(* CODESYS project MC500.project
   Title: MC500
   CompiledLibraryCompatibilityVersion: LeadSysStudio V3.5 SP15 Patch 4

Project tree, tasks and I/O mapping:
  Device : MC508, Leadshine Technology Co., Ltd., order no. 508101, version 3.5.15.40
      settings: RetainMode = 0; RetainStartAddr = 20480; RetainEndAddr = 524288; RetainSize = 524288
    application Application
      libraries: Standard, * (System); VisuDialogs, * (System)
      task EtherCAT_Master_Leadshine_A (cyclic, interval 2000 µs, priority 0) calls EtherCAT_Master_Leadshine_A.EtherCAT_Task [EtherCAT_Master_Leadshine_A.EtherCAT_Task], main
      program main [ST]: initialize, motion, gear, io, tap, index, work, WRAP
      visualisation Visualization
      trace Trace (task EtherCAT_Master_Leadshine_A): main.gear_data.trace_master, main.gear_data.trace_slave, main.gear_data.trace_delta
      data type GearData
      data type IOTestData
      data type TapData
      data type IndexData
      data type WorkData
      Symbols
      data type ButtonData
    Device Diagnose
    Network Configuration
      LocalBus Config
    Resource Usage
    SoftMotion General Axis Pool
    High_Speed_IO_Module : High Speed IO, Leadshine Technology Co., Ltd., version 3.5.15.40
        unmapped channels: Genral_IO_IN, Genral_IO_Out
    LocalBus_Master_Module : LocalBus Master, Leadshine Technology Co., Ltd., version 3.5.15.40
    EtherCAT_Master_Leadshine_A : EtherCAT Master SoftMotion, 3S - Smart Software Solutions GmbH, version 3.5.15.30
        settings: MasterCycleTime = 2000; NetworkName = 'ecat'; SelectNetworkByName = False; SrcAddress1 = 10; SrcAddress2 = 889192738
      AxisX : XINJE-DS5C EtherCAT(CoE) Drive Rev2.0 v3.7.30, Xinje Electronics, Inc., order no. XINJE-DS5C CoE Drive Rev2.0, version Revision=16#02040608
          settings: Number of Inputs = 6; Number of Infos about Inputs = 6; EnableExpertSettings = True; StationAlias = 1; DeviceIdenticationADO = 0; DeviceIdenticationMode = 0; Sync.Length = 17; FMMU.Length = 17; DC sync0 cycletime = 2000; DC sync1 cycletime = 2000; Number of SDO = 5; Interpolation time period.Value = 2; Homing method.Index = 16#0000; Homing method.Subindex = 16#00; Homing method.Size = 0; Homing method.AbortIfError = FALSE; Homing method.JumpToLine = FALSE; Homing method.Line = 0; Homing method.CompleteAccess = False; Homing method.Index = 16#0000; Homing method.Subindex = 16#00; Homing method.Size = 0; Homing method.AbortIfError = FALSE; Homing method.JumpToLine = FALSE; Homing method.Line = 0; Homing method.CompleteAccess = False; RxTxPdo.NumberofEntries = 6; RxTxPdo.Index = 16#1A00; RxTxPdo.DependOnSlot = False; RxTxPdo.DependOnSlotGroup = False; RxTxPdo.OverwrittenByModule = False; Status Word.Offset = 0; Status Word.DependOnSlot = False; Status Word.DependOnSlotGroup = False; ActualPosition.Offset = 0; ActualPosition.DependOnSlot = False; ActualPosition.DependOnSlotGroup = False; Velocity actual value.Offset = 0; Velocity actual value.DependOnSlot = False; Velocity actual value.DependOnSlotGroup = False;
            ActualTorque.Offset = 0; ActualTorque.DependOnSlot = False; ActualTorque.DependOnSlotGroup = False; ModeOfOperationDisplay.Offset = 0; ModeOfOperationDisplay.DependOnSlot = False; ModeOfOperationDisplay.DependOnSlotGroup = False; Index = 16#5000; SubIndex = 0; Size = 32; Offset = 0; DependOnSlot = False; DependOnSlotGroup = False; Status Word.Default = ''; Status Word.Comment = ''; ActualPosition.Default = ''; ActualPosition.Comment = ''; Velocity actual value.Default = ''; Velocity actual value.Comment = ''; ActualTorque.Default = ''; ActualTorque.Comment = ''; ModeOfOperationDisplay.Default = ''; ModeOfOperationDisplay.Comment = ''; Name = 'Encode Single Position'; DataType = 'DINT'; Default = ''; Comment = ''
          unmapped channels: Control Word, TargetPosition, TargetVelocity, TargetTorque, ModeOfOperation, Status Word, ActualPosition, Velocity actual value, %IW8 ActualTorque, ModeOfOperationDisplay, %ID5 Encode Single Position
        AX : Axis, 3S - Smart Software Solutions GmbH, order no. 0, version 4.6.1.0
            settings: wDriveID = 0; dwRatioTechUnitsDenom = 16384; iRatioTechUnitsNum = 625; fSWLimitPositive = 5000.0; Number of pulses for one revolution = 1; The displacement for one revolution of the workbench = 1; Gear ratio molecule = 131072; Gear ratio denominator = 5000; ScalingIncs = 1; ScalingMotorTurns2 = 131072; ScalingGearOutput1 = 5000; AdrOffset_8010 = 4; BitOffset_8010 = 0; BitLength_8010 = 16; Address_8010 = '%QW2'; Type_8010 = 'UINT'; AddressPointer_8010 = ADR(%QW2); AdrOffset_8020 = 8; BitOffset_8020 = 0; BitLength_8020 = 32; Address_8020 = '%QD2'; Type_8020 = 'DINT'; AddressPointer_8020 = ADR(%QD2); AdrOffset_8030 = 12; BitOffset_8030 = 0; BitLength_8030 = 32; Address_8030 = '%QD3'; Type_8030 = 'DINT'; AddressPointer_8030 = ADR(%QD3); AdrOffset_8040 = 16; BitOffset_8040 = 0; BitLength_8040 = 16; Address_8040 = '%QW8'; Type_8040 = 'INT'; AddressPointer_8040 = ADR(%QW8); AdrOffset_8050 = 18; BitOffset_8050 = 0; BitLength_8050 = 8; Address_8050 = '%QB18'; Type_8050 = 'SINT';
              AddressPointer_8050 = ADR(%QB18); AdrOffset_8060 = 4294967295; BitOffset_8060 = 0; BitLength_8060 = 0; Address_8060 = ''; Type_8060 = ''; AddressPointer_8060 = 0; AdrOffset_8070 = 4294967295; BitOffset_8070 = 0; BitLength_8070 = 0; Address_8070 = ''; Type_8070 = ''; AddressPointer_8070 = 0; AdrOffset_8080 = 4294967295; BitOffset_8080 = 0; BitLength_8080 = 0; Address_8080 = ''; Type_8080 = ''; AddressPointer_8080 = 0; AdrOffset_8090 = 4294967295; BitOffset_8090 = 0; BitLength_8090 = 0; Address_8090 = ''; Type_8090 = ''; AddressPointer_8090 = 0; AdrOffset_8510 = 4; BitOffset_8510 = 0; BitLength_8510 = 16; Address_8510 = '%IW2'; Type_8510 = 'UINT'; AddressPointer_8510 = ADR(%IW2); AdrOffset_8520 = 8; BitOffset_8520 = 0; BitLength_8520 = 32; Address_8520 = '%ID2'; Type_8520 = 'DINT'; AddressPointer_8520 = ADR(%ID2); AdrOffset_8530 = 12; BitOffset_8530 = 0; BitLength_8530 = 32;
              Address_8530 = '%ID3'; Type_8530 = 'DINT'; AddressPointer_8530 = ADR(%ID3); AdrOffset_8540 = 16; BitOffset_8540 = 0; BitLength_8540 = 16; Address_8540 = '%IW8'; Type_8540 = 'INT'; AddressPointer_8540 = ADR(%IW8); AdrOffset_8550 = 18; BitOffset_8550 = 0; BitLength_8550 = 8; Address_8550 = '%IB18'; Type_8550 = 'SINT'; AddressPointer_8550 = ADR(%IB18); AdrOffset_8560 = 4294967295; BitOffset_8560 = 0; BitLength_8560 = 0; Address_8560 = ''; Type_8560 = ''; AddressPointer_8560 = 0; AdrOffset_8570 = 4294967295; BitOffset_8570 = 0; BitLength_8570 = 0; Address_8570 = ''; Type_8570 = ''; AddressPointer_8570 = 0; AdrOffset_8580 = 4294967295; BitOffset_8580 = 0; BitLength_8580 = 0; Address_8580 = ''; Type_8580 = ''; AddressPointer_8580 = 0; AdrOffset_8590 = 4294967295; BitOffset_8590 = 0; BitLength_8590 = 0; Address_8590 = ''; Type_8590 = ''; AddressPointer_8590 = 0; AdrOffset_8600 = 4294967295;
              BitOffset_8600 = 0; BitLength_8600 = 0; Address_8600 = ''; Type_8600 = ''; AddressPointer_8600 = 0; AdrOffset_8600 = 4294967295; BitOffset_8600 = 0; BitLength_8600 = 0; Address_8610 = ''; Type_8610 = ''; AddressPointer_8610 = 0; AdrOffset_8620 = 4294967295; BitOffset_8620 = 0; BitLength_8620 = 0; Address_8620 = ''; Type_8620 = ''; AddressPointer_8620 = 0
      AxisY : XINJE-DS5C EtherCAT(CoE) Drive Rev2.0 v3.7.30, Xinje Electronics, Inc., order no. XINJE-DS5C CoE Drive Rev2.0, version Revision=16#02040608
          settings: Number of Inputs = 6; Number of Infos about Inputs = 6; EnableExpertSettings = True; StationAlias = 2; DeviceIdenticationADO = 0; DeviceIdenticationMode = 0; Sync.Length = 17; FMMU.Length = 17; DC sync0 cycletime = 2000; DC sync1 cycletime = 2000; Number of SDO = 5; Interpolation time period.Value = 2; Homing method.Index = 16#0000; Homing method.Subindex = 16#00; Homing method.Size = 0; Homing method.AbortIfError = FALSE; Homing method.JumpToLine = FALSE; Homing method.Line = 0; Homing method.CompleteAccess = False; Homing method.Index = 16#0000; Homing method.Subindex = 16#00; Homing method.Size = 0; Homing method.AbortIfError = FALSE; Homing method.JumpToLine = FALSE; Homing method.Line = 0; Homing method.CompleteAccess = False; RxTxPdo.NumberofEntries = 6; RxTxPdo.Index = 16#1A00; RxTxPdo.DependOnSlot = False; RxTxPdo.DependOnSlotGroup = False; RxTxPdo.OverwrittenByModule = False; Status Word.Offset = 0; Status Word.DependOnSlot = False; Status Word.DependOnSlotGroup = False; ActualPosition.Offset = 0; ActualPosition.DependOnSlot = False; ActualPosition.DependOnSlotGroup = False; Velocity actual value.Offset = 0; Velocity actual value.DependOnSlot = False; Velocity actual value.DependOnSlotGroup = False;
            ActualTorque.Offset = 0; ActualTorque.DependOnSlot = False; ActualTorque.DependOnSlotGroup = False; ModeOfOperationDisplay.Offset = 0; ModeOfOperationDisplay.DependOnSlot = False; ModeOfOperationDisplay.DependOnSlotGroup = False; Index = 16#5000; SubIndex = 0; Size = 32; Offset = 0; DependOnSlot = False; DependOnSlotGroup = False; Status Word.Default = ''; Status Word.Comment = ''; ActualPosition.Default = ''; ActualPosition.Comment = ''; Velocity actual value.Default = ''; Velocity actual value.Comment = ''; ActualTorque.Default = ''; ActualTorque.Comment = ''; ModeOfOperationDisplay.Default = ''; ModeOfOperationDisplay.Comment = ''; Name = 'Encode Single Position'; DataType = 'DINT'; Default = ''; Comment = ''
          unmapped channels: Control Word, TargetPosition, TargetVelocity, TargetTorque, ModeOfOperation, Status Word, ActualPosition, Velocity actual value, %IW18 ActualTorque, ModeOfOperationDisplay, %ID10 Encode Single Position
        AY : Axis, 3S - Smart Software Solutions GmbH, order no. 0, version 4.6.1.0
            settings: dwRatioTechUnitsDenom = 16384; iRatioTechUnitsNum = 125; Number of pulses for one revolution = 1; The displacement for one revolution of the workbench = 1; Gear ratio molecule = 131072; Gear ratio denominator = 1000; ScalingIncs = 1; ScalingMotorTurns2 = 131072; ScalingGearOutput1 = 1000; AdrOffset_8010 = 20; BitOffset_8010 = 0; BitLength_8010 = 16; Address_8010 = '%QW10'; Type_8010 = 'UINT'; AddressPointer_8010 = ADR(%QW10); AdrOffset_8020 = 24; BitOffset_8020 = 0; BitLength_8020 = 32; Address_8020 = '%QD6'; Type_8020 = 'DINT'; AddressPointer_8020 = ADR(%QD6); AdrOffset_8030 = 28; BitOffset_8030 = 0; BitLength_8030 = 32; Address_8030 = '%QD7'; Type_8030 = 'DINT'; AddressPointer_8030 = ADR(%QD7); AdrOffset_8040 = 32; BitOffset_8040 = 0; BitLength_8040 = 16; Address_8040 = '%QW16'; Type_8040 = 'INT'; AddressPointer_8040 = ADR(%QW16); AdrOffset_8050 = 34; BitOffset_8050 = 0; BitLength_8050 = 8; Address_8050 = '%QB34'; Type_8050 = 'SINT'; AddressPointer_8050 = ADR(%QB34); AdrOffset_8060 = 4294967295;
              BitOffset_8060 = 0; BitLength_8060 = 0; Address_8060 = ''; Type_8060 = ''; AddressPointer_8060 = 0; AdrOffset_8070 = 4294967295; BitOffset_8070 = 0; BitLength_8070 = 0; Address_8070 = ''; Type_8070 = ''; AddressPointer_8070 = 0; AdrOffset_8080 = 4294967295; BitOffset_8080 = 0; BitLength_8080 = 0; Address_8080 = ''; Type_8080 = ''; AddressPointer_8080 = 0; AdrOffset_8090 = 4294967295; BitOffset_8090 = 0; BitLength_8090 = 0; Address_8090 = ''; Type_8090 = ''; AddressPointer_8090 = 0; AdrOffset_8510 = 24; BitOffset_8510 = 0; BitLength_8510 = 16; Address_8510 = '%IW12'; Type_8510 = 'UINT'; AddressPointer_8510 = ADR(%IW12); AdrOffset_8520 = 28; BitOffset_8520 = 0; BitLength_8520 = 32; Address_8520 = '%ID7'; Type_8520 = 'DINT'; AddressPointer_8520 = ADR(%ID7); AdrOffset_8530 = 32; BitOffset_8530 = 0; BitLength_8530 = 32; Address_8530 = '%ID8'; Type_8530 = 'DINT';
              AddressPointer_8530 = ADR(%ID8); AdrOffset_8540 = 36; BitOffset_8540 = 0; BitLength_8540 = 16; Address_8540 = '%IW18'; Type_8540 = 'INT'; AddressPointer_8540 = ADR(%IW18); AdrOffset_8550 = 38; BitOffset_8550 = 0; BitLength_8550 = 8; Address_8550 = '%IB38'; Type_8550 = 'SINT'; AddressPointer_8550 = ADR(%IB38); AdrOffset_8560 = 4294967295; BitOffset_8560 = 0; BitLength_8560 = 0; Address_8560 = ''; Type_8560 = ''; AddressPointer_8560 = 0; AdrOffset_8570 = 4294967295; BitOffset_8570 = 0; BitLength_8570 = 0; Address_8570 = ''; Type_8570 = ''; AddressPointer_8570 = 0; AdrOffset_8580 = 4294967295; BitOffset_8580 = 0; BitLength_8580 = 0; Address_8580 = ''; Type_8580 = ''; AddressPointer_8580 = 0; AdrOffset_8590 = 4294967295; BitOffset_8590 = 0; BitLength_8590 = 0; Address_8590 = ''; Type_8590 = ''; AddressPointer_8590 = 0; AdrOffset_8600 = 4294967295; BitOffset_8600 = 0; BitLength_8600 = 0;
              Address_8600 = ''; Type_8600 = ''; AddressPointer_8600 = 0; AdrOffset_8600 = 4294967295; BitOffset_8600 = 0; BitLength_8600 = 0; Address_8610 = ''; Type_8610 = ''; AddressPointer_8610 = 0; AdrOffset_8620 = 4294967295; BitOffset_8620 = 0; BitLength_8620 = 0; Address_8620 = ''; Type_8620 = ''; AddressPointer_8620 = 0
      AxisZ : XINJE-DS5C1 EtherCAT(CoE) Drive Rev4.0 v3.7.70, Xinje Electronics, Inc., order no. XINJE-DS5C1 CoE Drive Rev4.0, version Revision=16#20201207
          settings: Number of Inputs = 6; Number of Infos about Inputs = 6; EnableExpertSettings = True; StationAlias = 3; DeviceIdenticationADO = 0; DeviceIdenticationMode = 0; Sync.Length = 17; FMMU.Length = 17; DC sync0 cycletime = 2000; DC sync1 cycletime = 2000; Number of SDO = 6; Interpolation time period.Value = 2; Homing method.Index = 16#0000; Homing method.Subindex = 16#00; Homing method.Size = 0; Homing method.AbortIfError = FALSE; Homing method.JumpToLine = FALSE; Homing method.Line = 0; Homing method.CompleteAccess = False; Homing method.Index = 16#0000; Homing method.Subindex = 16#00; Homing method.Size = 0; Homing method.AbortIfError = FALSE; Homing method.JumpToLine = FALSE; Homing method.Line = 0; Homing method.CompleteAccess = False; Homing method.Index = 16#0000; Homing method.Subindex = 16#00; Homing method.Size = 0; Homing method.AbortIfError = FALSE; Homing method.JumpToLine = FALSE; Homing method.Line = 0; Homing method.CompleteAccess = False; RxTxPdo.NumberofEntries = 6; RxTxPdo.Index = 16#1A00; RxTxPdo.DependOnSlot = False; RxTxPdo.DependOnSlotGroup = False; RxTxPdo.OverwrittenByModule = False; Status Word.Offset = 0; Status Word.DependOnSlot = False;
            Status Word.DependOnSlotGroup = False; ActualPosition.Offset = 0; ActualPosition.DependOnSlot = False; ActualPosition.DependOnSlotGroup = False; Velocity actual value.Offset = 0; Velocity actual value.DependOnSlot = False; Velocity actual value.DependOnSlotGroup = False; ActualTorque.Offset = 0; ActualTorque.DependOnSlot = False; ActualTorque.DependOnSlotGroup = False; ModeOfOperationDisplay.Offset = 0; ModeOfOperationDisplay.DependOnSlot = False; ModeOfOperationDisplay.DependOnSlotGroup = False; Index = 16#5000; SubIndex = 0; Size = 32; Offset = 0; DependOnSlot = False; DependOnSlotGroup = False; Status Word.Default = ''; Status Word.Comment = ''; ActualPosition.Default = ''; ActualPosition.Comment = ''; Velocity actual value.Default = ''; Velocity actual value.Comment = ''; ActualTorque.Default = ''; ActualTorque.Comment = ''; ModeOfOperationDisplay.Default = ''; ModeOfOperationDisplay.Comment = ''; Name = 'Encode Single Position'; DataType = 'DINT'; Default = ''; Comment = ''
          unmapped channels: Control Word, TargetPosition, TargetVelocity, TargetTorque, ModeOfOperation, Status Word, ActualPosition, Velocity actual value, %IW28 ActualTorque, ModeOfOperationDisplay, %ID15 Encode Single Position
        AZ : Axis, 3S - Smart Software Solutions GmbH, order no. 0, version 4.6.1.0
            settings: wDriveID = 2; dwRatioTechUnitsDenom = 1; iMovementType = 0; fPositionPeriod = 131072; Number of pulses for one revolution = 1; The displacement for one revolution of the workbench = 1; Gear ratio molecule = 1; Gear ratio denominator = 1; ScalingIncs = 1; AdrOffset_8010 = 36; BitOffset_8010 = 0; BitLength_8010 = 16; Address_8010 = '%QW18'; Type_8010 = 'UINT'; AddressPointer_8010 = ADR(%QW18); AdrOffset_8020 = 40; BitOffset_8020 = 0; BitLength_8020 = 32; Address_8020 = '%QD10'; Type_8020 = 'DINT'; AddressPointer_8020 = ADR(%QD10); AdrOffset_8030 = 44; BitOffset_8030 = 0; BitLength_8030 = 32; Address_8030 = '%QD11'; Type_8030 = 'DINT'; AddressPointer_8030 = ADR(%QD11); AdrOffset_8040 = 48; BitOffset_8040 = 0; BitLength_8040 = 16; Address_8040 = '%QW24'; Type_8040 = 'INT'; AddressPointer_8040 = ADR(%QW24); AdrOffset_8050 = 50; BitOffset_8050 = 0; BitLength_8050 = 8; Address_8050 = '%QB50'; Type_8050 = 'SINT'; AddressPointer_8050 = ADR(%QB50); AdrOffset_8060 = 4294967295;
              BitOffset_8060 = 0; BitLength_8060 = 0; Address_8060 = ''; Type_8060 = ''; AddressPointer_8060 = 0; AdrOffset_8070 = 4294967295; BitOffset_8070 = 0; BitLength_8070 = 0; Address_8070 = ''; Type_8070 = ''; AddressPointer_8070 = 0; AdrOffset_8080 = 4294967295; BitOffset_8080 = 0; BitLength_8080 = 0; Address_8080 = ''; Type_8080 = ''; AddressPointer_8080 = 0; AdrOffset_8090 = 4294967295; BitOffset_8090 = 0; BitLength_8090 = 0; Address_8090 = ''; Type_8090 = ''; AddressPointer_8090 = 0; AdrOffset_8510 = 44; BitOffset_8510 = 0; BitLength_8510 = 16; Address_8510 = '%IW22'; Type_8510 = 'UINT'; AddressPointer_8510 = ADR(%IW22); AdrOffset_8520 = 48; BitOffset_8520 = 0; BitLength_8520 = 32; Address_8520 = '%ID12'; Type_8520 = 'DINT'; AddressPointer_8520 = ADR(%ID12); AdrOffset_8530 = 52; BitOffset_8530 = 0; BitLength_8530 = 32; Address_8530 = '%ID13'; Type_8530 = 'DINT';
              AddressPointer_8530 = ADR(%ID13); AdrOffset_8540 = 56; BitOffset_8540 = 0; BitLength_8540 = 16; Address_8540 = '%IW28'; Type_8540 = 'INT'; AddressPointer_8540 = ADR(%IW28); AdrOffset_8550 = 58; BitOffset_8550 = 0; BitLength_8550 = 8; Address_8550 = '%IB58'; Type_8550 = 'SINT'; AddressPointer_8550 = ADR(%IB58); AdrOffset_8560 = 4294967295; BitOffset_8560 = 0; BitLength_8560 = 0; Address_8560 = ''; Type_8560 = ''; AddressPointer_8560 = 0; AdrOffset_8570 = 4294967295; BitOffset_8570 = 0; BitLength_8570 = 0; Address_8570 = ''; Type_8570 = ''; AddressPointer_8570 = 0; AdrOffset_8580 = 4294967295; BitOffset_8580 = 0; BitLength_8580 = 0; Address_8580 = ''; Type_8580 = ''; AddressPointer_8580 = 0; AdrOffset_8590 = 4294967295; BitOffset_8590 = 0; BitLength_8590 = 0; Address_8590 = ''; Type_8590 = ''; AddressPointer_8590 = 0; AdrOffset_8600 = 4294967295; BitOffset_8600 = 0; BitLength_8600 = 0;
              Address_8600 = ''; Type_8600 = ''; AddressPointer_8600 = 0; AdrOffset_8600 = 4294967295; BitOffset_8600 = 0; BitLength_8600 = 0; Address_8610 = ''; Type_8610 = ''; AddressPointer_8610 = 0; AdrOffset_8620 = 4294967295; BitOffset_8620 = 0; BitLength_8620 = 0; Address_8620 = ''; Type_8620 = ''; AddressPointer_8620 = 0
  text list GlobalTextList
*)

// Device/Application/GearData
TYPE GearData :
STRUCT
	state: INT;
	ratio_target: LREAL;
	ratio: LREAL;
	ratio_array: ARRAY[0..14] OF LREAL;
	ratio_array_index: INT;
	reset_gear_timer: TON;
	trace_master: LREAL;
	trace_slave: LREAL;
	trace_delta: LREAL;
END_STRUCT
END_TYPE

// Device/Application/IOTestData
TYPE IOTestData :
STRUCT
	out: WORD;
	out_timer: TON;
END_STRUCT
END_TYPE

// Device/Application/TapData
TYPE TapData :
STRUCT
	state: INT;
	home_torque: INT;
	home_feed_back: LREAL;
	home_feed_forward: LREAL;
	home_offset: LREAL;
	start_position: LREAL;
	end_position: LREAL;
	feed_rpm: LREAL;
	end_delay: INT;
	end_timer: TON;
	gear_type: INT;
END_STRUCT
END_TYPE

// Device/Application/IndexData
TYPE IndexData :
STRUCT
	state: INT;
	slot_count: INT;
	slot_index: INT;
	slot_index_nearest: INT;
	real_position: LREAL;
	soft_position: LREAL;
	target_position: LREAL;
	offset: LREAL;
	ecd_sing: LREAL;
	ecd_reso: LREAL;
	end_delay: INT;
	end_timer: TON;
	feed_rpm: LREAL;
	is_home_ing: BOOL;
	vibrate_distance: LREAL;
END_STRUCT
END_TYPE

// Device/Application/WorkData
TYPE WorkData :
STRUCT
	state: INT;
	stop_state: INT;
	end_delay: INT;
	end_timer: TON;
END_STRUCT
END_TYPE

// Device/Application/ButtonData
TYPE ButtonData :
STRUCT
	on: BOOL;
	off: BOOL;
END_STRUCT
END_TYPE

// Device/Application/main
PROGRAM main
VAR
	state: INT;
	AX_power: MC_Power;
	AY_power: MC_Power;
	AZ_power: MC_Power;
	AX_status: MC_ReadStatus;
	AY_status: MC_ReadStatus;
	AZ_status: MC_ReadStatus;
	AZ_stop: MC_Stop;
	AX_reset: MC_Reset;
	AY_reset: MC_Reset;
	AZ_reset: MC_Reset;
	AX_set_position: MC_SetPosition;
	AY_set_position: MC_SetPosition;
	AZ_set_position: MC_SetPosition;
	AZ_mabs: MC_MoveAbsolute;
	AX_read: SMC3_ETC_ReadParameter_CoE;
	AY_read: SMC3_ETC_ReadParameter_CoE;
	AZ_read: SMC3_ETC_ReadParameter_CoE;
	AX_write: SMC3_ETC_WriteParameter_CoE;
	AY_write: SMC3_ETC_WriteParameter_CoE;
	AZ_write: SMC3_ETC_WriteParameter_CoE;
	AX_follow: SMC_FollowPosition;
	AY_follow: SMC_FollowPosition;
	gear_data: GearData;
	AX_torque AT %IW8: INT;
	AY_torque AT %IW18: INT;
	AZ_torque AT %IW28: INT;
	AX_encoder_single AT %ID5: DINT;
	AY_encoder_single AT %ID10: DINT;
	AZ_encoder_single AT %ID15: DINT;
	AX_encoder_resolution: DINT;
	AY_encoder_resolution: DINT;
	AZ_encoder_resolution: DINT;
	io_test_data: IOTestData;
	index_data: IndexData;
	tap_data: TapData;
	work_data: WorkData;
	button_data: ButtonData;
END_VAR

CASE state OF
    0:
		initialize();
		state := state + 1;
	1:
		IF AX.wCommunicationState = 100 AND AY.wCommunicationState = 100 AND AZ.wCommunicationState = 100 THEN
			AX_power.Enable := TRUE;
			AY_power.Enable := TRUE;
			AZ_power.Enable := TRUE;
			AX_status.Enable := TRUE;
			AY_status.Enable := TRUE;
			AZ_status.Enable := TRUE;
			AX_power.bDriveStart := TRUE;
			AY_power.bDriveStart := TRUE;
			AZ_power.bDriveStart := TRUE;
			AX_power.bRegulatorOn := FALSE;
			AY_power.bRegulatorOn := FALSE;
			AZ_power.bRegulatorOn := FALSE;
			state := state + 1;
		END_IF
	2:
		gear_data.ratio_array_index := 0;
		work_data.state := 1;
		state := state + 1;
	3:
		io();
END_CASE

IF state >= 2 THEN
	gear();
	motion();
	index();
	tap();
	work();
END_IF

ACTION initialize:
gear_data.ratio_array_index := 0;
gear_data.ratio_array[0] := 0.5;
gear_data.ratio_array[1] := 1.0;
gear_data.ratio_array[2] := 1.5;
gear_data.ratio_array[3] := 2.0;
gear_data.ratio_array[4] := 2.5;
gear_data.ratio_array[5] := 3.0;
gear_data.ratio_array[6] := 3.5;
gear_data.ratio_array[7] := 4.0;
gear_data.ratio_array[8] := 4.5;
gear_data.ratio_array[9] := 5.0;
gear_data.ratio_array[10] := 10.0;
gear_data.ratio_array[11] := 15.0;
gear_data.ratio_array[12] := 20.0;
gear_data.ratio_array[13] := 25.0;
gear_data.ratio_array[14] := 50.0;
state := 0;
index_data.state := 0;
index_data.end_delay := 100;
index_data.slot_count := 8;
index_data.feed_rpm := 60.0;
index_data.vibrate_distance := 1.0 / 64.0;
tap_data.state := 0;
tap_data.end_delay := 25;
tap_data.home_torque := 200;
tap_data.home_feed_back := 2000.0;
tap_data.home_feed_forward := 3000.0;
tap_data.home_offset := 10_000.0;
tap_data.start_position := tap_data.home_offset;
tap_data.end_position := tap_data.home_offset + 7_000.0;
tap_data.feed_rpm := 800.0;
tap_data.gear_type := 1;
work_data.state := 0;
work_data.stop_state := 0;
work_data.end_delay := 25;
button_data.on := FALSE;
button_data.off := FALSE;
END_ACTION

ACTION motion:
IF AX.bCommunication AND AY.bCommunication AND AZ.bCommunication THEN
	//power
	AX_power( Axis:= AX, Enable:= , bRegulatorOn:= , bDriveStart:= , Status=> , bRegulatorRealState=> , bDriveStartRealState=> , Busy=> , Error=> , ErrorID=> );
	AY_power( Axis:= AY, Enable:= , bRegulatorOn:= , bDriveStart:= , Status=> , bRegulatorRealState=> , bDriveStartRealState=> , Busy=> , Error=> , ErrorID=> );
	AZ_power( Axis:= AZ, Enable:= , bRegulatorOn:= , bDriveStart:= , Status=> , bRegulatorRealState=> , bDriveStartRealState=> , Busy=> , Error=> , ErrorID=> );
	//status
	AX_status( Axis:= AX, Enable:= , Valid=> , Busy=> , Error=> , ErrorID=> , Disabled=> , Errorstop=> , Stopping=> , StandStill=> , DiscreteMotion=> , ContinuousMotion=> , SynchronizedMotion=> , Homing=> , ConstantVelocity=> , Accelerating=> , Decelerating=> , FBErrorOccured=> );
	AY_status( Axis:= AY, Enable:= , Valid=> , Busy=> , Error=> , ErrorID=> , Disabled=> , Errorstop=> , Stopping=> , StandStill=> , DiscreteMotion=> , ContinuousMotion=> , SynchronizedMotion=> , Homing=> , ConstantVelocity=> , Accelerating=> , Decelerating=> , FBErrorOccured=> );
	AZ_status( Axis:= AZ, Enable:= , Valid=> , Busy=> , Error=> , ErrorID=> , Disabled=> , Errorstop=> , Stopping=> , StandStill=> , DiscreteMotion=> , ContinuousMotion=> , SynchronizedMotion=> , Homing=> , ConstantVelocity=> , Accelerating=> , Decelerating=> , FBErrorOccured=> );
	//stop
	AZ_stop( Axis:= AZ, Execute:= , Deceleration:= , Jerk:= , Done=> , Busy=> , Error=> , ErrorID=> );
	//reset
	AX_reset( Axis:= AX, Execute:= , Done=> , Busy=> , Error=> , ErrorID=> );
	AY_reset( Axis:= AY, Execute:= , Done=> , Busy=> , Error=> , ErrorID=> );
	AZ_reset( Axis:= AZ, Execute:= , Done=> , Busy=> , Error=> , ErrorID=> );
	//set position
	AX_set_position( Axis:= AX, Execute:= , Position:= , Mode:= , Done=> , Busy=> , Error=> , ErrorID=> );
	AY_set_position( Axis:= AY, Execute:= , Position:= , Mode:= , Done=> , Busy=> , Error=> , ErrorID=> );
	AZ_set_position( Axis:= AZ, Execute:= , Position:= , Mode:= , Done=> , Busy=> , Error=> , ErrorID=> );
	//move absolute
	AZ_mabs( Axis:= AZ, Execute:= , Position:= , Velocity:= , Acceleration:= , Deceleration:= , Jerk:= , Direction:= , BufferMode:= , Done=> , Busy=> , Active=> , CommandAborted=> , Error=> , ErrorID=> );
	//read write
	AX_read( xExecute:= , xAbort:= , uiIndex:= , usiSubIndex:= , Axis:= AX, xDone=> , xBusy=> , xError=> , usiDataLength=> , dwValue=> , dwErrorCode=> , eError=> );
	AY_read( xExecute:= , xAbort:= , uiIndex:= , usiSubIndex:= , Axis:= AY, xDone=> , xBusy=> , xError=> , usiDataLength=> , dwValue=> , dwErrorCode=> , eError=> );
	AZ_read( xExecute:= , xAbort:= , uiIndex:= , usiSubIndex:= , Axis:= AZ, xDone=> , xBusy=> , xError=> , usiDataLength=> , dwValue=> , dwErrorCode=> , eError=> );
	AX_write( xExecute:= , xAbort:= , uiIndex:= , usiSubIndex:= , usiDataLength:= , dwValue:= , Axis:= AX, xDone=> , xBusy=> , xError=> , dwErrorCode=> , eError=> );
	AY_write( xExecute:= , xAbort:= , uiIndex:= , usiSubIndex:= , usiDataLength:= , dwValue:= , Axis:= AY, xDone=> , xBusy=> , xError=> , dwErrorCode=> , eError=> );
	AZ_write( xExecute:= , xAbort:= , uiIndex:= , usiSubIndex:= , usiDataLength:= , dwValue:= , Axis:= AZ, xDone=> , xBusy=> , xError=> , dwErrorCode=> , eError=> );
	//follow
	AX_follow( Axis:= AX, bExecute:= , fSetPosition:= , bBusy=> , bCommandAborted=> , bError=> , iErrorID=> );
	AY_follow( Axis:= AY, bExecute:= , fSetPosition:= , bBusy=> , bCommandAborted=> , bError=> , iErrorID=> );
END_IF
END_ACTION

ACTION gear:
gear_data.ratio_target := gear_data.ratio_array[gear_data.ratio_array_index];
gear_data.trace_master := AY.fActPosition;
gear_data.trace_slave := AX.fActPosition / gear_data.ratio;
gear_data.trace_delta := gear_data.trace_master - gear_data.trace_slave;
CASE gear_data.state OF
	0:
		gear_data.reset_gear_timer.IN := FALSE;
	1:
		AX_follow.bExecute := FALSE;
		AY_follow.bExecute := FALSE;
		AX_power.bRegulatorOn := FALSE;
		AY_power.bRegulatorOn := FALSE;
		gear_data.state := gear_data.state + 1;
	2:
		gear_data.reset_gear_timer(IN:= , PT:= , Q=> , ET=> );
		IF NOT gear_data.reset_gear_timer.IN THEN
			gear_data.reset_gear_timer.IN := TRUE;
			gear_data.reset_gear_timer.PT := INT_TO_TIME(100);
		END_IF
		IF gear_data.reset_gear_timer.Q THEN
			gear_data.reset_gear_timer.IN := FALSE;
			gear_data.state := gear_data.state + 1;
		END_IF
	3:
		IF AX_status.FBErrorOccured AND NOT AX_reset.Execute THEN
			AX_reset.Execute := TRUE;
		END_IF
		IF AY_status.FBErrorOccured AND NOT AY_reset.Execute THEN
			AY_reset.Execute := TRUE;
		END_IF
		gear_data.state := gear_data.state + 1;
	4:
		IF NOT (AX_status.FBErrorOccured OR AY_status.FBErrorOccured) THEN
			AX_reset.Execute := FALSE;
			AY_reset.Execute := FALSE;
			gear_data.state := gear_data.state + 1;
		END_IF
	5:
		gear_data.state := 0;
	//on x off y -> gear x to y
	101:
		AX_power.bRegulatorOn := TRUE;
		AY_power.bRegulatorOn := FALSE;
		gear_data.state := gear_data.state + 1;
	102:
		IF AX_power.Status AND NOT AY_power.Status THEN
			gear_data.ratio := gear_data.ratio_target;
			gear_data.state := gear_data.state + 1;
		END_IF
	103:
		AY_set_position.Position := AX.fActPosition / gear_data.ratio;
		AY_set_position.Execute := TRUE;
		gear_data.state := gear_data.state + 1;
	104:
		IF AY_set_position.Done THEN
			AY_set_position.Execute := FALSE;
			gear_data.state := gear_data.state + 1;
		END_IF
	105:
		AX_follow.fSetPosition := AY.fActPosition * gear_data.ratio;
		AX_follow.bExecute := TRUE;
		gear_data.state := 200;
	200:
		AX_follow.fSetPosition := AY.fActPosition * gear_data.ratio;
	
	//on x on y -> gear x to y follow position
	201:
		AX_power.bRegulatorOn := TRUE;
		AY_power.bRegulatorOn := TRUE;
		gear_data.state := gear_data.state + 1;
	202:
		IF AX_power.Status AND AY_power.Status THEN
			gear_data.ratio := gear_data.ratio_target;
			gear_data.state := gear_data.state + 1;
		END_IF
	203:
		AY_set_position.Position := AX.fActPosition / gear_data.ratio;
		AY_set_position.Execute := TRUE;
		gear_data.state := gear_data.state + 1;
	204:
		IF AY_set_position.Done THEN
			AY_set_position.Execute := FALSE;
			gear_data.state := gear_data.state + 1;
		END_IF
	205:
		AX_follow.fSetPosition := AY.fActPosition * gear_data.ratio;
		AY_follow.fSetPosition := AY.fActPosition;
		AX_follow.bExecute := TRUE;
		AY_follow.bExecute := TRUE;
		gear_data.state := 300;
	300:
		AX_follow.fSetPosition := AY_follow.fSetPosition * gear_data.ratio;
END_CASE
END_ACTION

ACTION io:
//input
IF button_data.on AND work_data.state = 0 THEN
	work_data.state := 101;
	button_data.on := FALSE;
END_IF
IF button_data.on AND work_data.state = 200 THEN
	work_data.state := 201;
END_IF
IF button_data.off THEN
	work_data.state := 1;
	button_data.off := FALSE;
	button_data.on := FALSE;
END_IF
//output
io_test_data.out_timer(IN:= , PT:= , Q=> , ET=> );
IF NOT io_test_data.out_timer.IN THEN
	io_test_data.out_timer.IN := TRUE;
	io_test_data.out_timer.PT := INT_TO_TIME(50);
END_IF
IF io_test_data.out_timer.Q THEN
	io_test_data.out := io_test_data.out * 2;
	IF io_test_data.out = 0 THEN
		io_test_data.out := 1;
	END_IF
	io_test_data.out_timer.IN := FALSE;
	%QW0 := io_test_data.out;
END_IF
END_ACTION

ACTION tap:
CASE tap_data.state OF
	0:
		tap_data.end_timer.IN := FALSE;
	//home
	1:
		gear_data.state := 1;
		tap_data.state := tap_data.state + 1;
	2:
		IF gear_data.state = 0 THEN
			gear_data.state := 201;
			tap_data.state := tap_data.state + 1;
		END_IF
	3:
		IF gear_data.state = 300 THEN
			tap_data.state := tap_data.state + 1;
		END_IF
	4:
		AY_follow.fSetPosition := AY_follow.fSetPosition - 5.0;
		IF ABS(AX_torque) > tap_data.home_torque THEN
			gear_data.state := 1;
			tap_data.state := tap_data.state + 1;
		END_IF
	5:
		IF gear_data.state = 0 THEN
			AX_set_position.Position := 0.0;
			AY_set_position.Position := 0.0;
			AX_set_position.Execute := TRUE;
			AY_set_position.Execute := TRUE;
			tap_data.state := tap_data.state + 1;
		END_IF
	6:
		IF AX_set_position.Done AND AY_set_position.Done THEN
			AX_set_position.Execute := FALSE;
			AY_set_position.Execute := FALSE;
			gear_data.state := 201;
			tap_data.state := tap_data.state + 1;
		END_IF
	7:
		IF gear_data.state = 300 THEN
			tap_data.state := tap_data.state + 1;
		END_IF
	8:
		AY_follow.fSetPosition := AY_follow.fSetPosition + 5.0;
		IF AX.fActPosition >= tap_data.start_position THEN
			tap_data.state := 100;
		END_IF
	//tap
    101:
		tap_data.state := tap_data.state + 1;
	102:
		AY_follow.fSetPosition := AY_follow.fSetPosition + 10.0;
		IF AX.fActPosition >= tap_data.end_position THEN
			tap_data.state := tap_data.state + 1;
		END_IF
	103:
		tap_data.state := tap_data.state + 1;
	104:
		AY_follow.fSetPosition := AY_follow.fSetPosition - 10.0;
		IF AX.fActPosition <= tap_data.start_position THEN
			tap_data.state := tap_data.state + 1;
		END_IF
	105:
		tap_data.end_timer(IN:= , PT:= , Q=> , ET=> );
		IF NOT tap_data.end_timer.IN THEN
			tap_data.end_timer.IN := TRUE;
			tap_data.end_timer.PT := INT_TO_TIME(tap_data.end_delay);
		END_IF
		IF tap_data.end_timer.Q THEN
			tap_data.state := 100;
			tap_data.end_timer.IN := FALSE;
		END_IF
END_CASE
END_ACTION

ACTION index:
index_data.ecd_sing := DINT_TO_LREAL(AZ_encoder_single);
IF AZ_encoder_resolution > 0 THEN
	index_data.ecd_reso := DINT_TO_LREAL(AZ_encoder_resolution);
	index_data.real_position := index_data.ecd_sing / index_data.ecd_reso;
	index_data.slot_index_nearest := LREAL_TO_INT(index_data.real_position * index_data.slot_count) MOD index_data.slot_count;
END_IF
CASE index_data.state OF
	0:
		index_data.end_timer.IN := FALSE;
	//home
    1:
		AZ_power.bRegulatorOn := TRUE;
		AZ_read.uiIndex := 16#608F;
		AZ_read.usiSubIndex := 1;
		AZ_read.xExecute := TRUE;
		index_data.state := index_data.state + 1;
	2:
		IF AZ_read.xDone THEN
			AZ_read.xExecute := FALSE;
			AZ_encoder_resolution := DWORD_TO_DINT(AZ_read.dwValue);
			index_data.state := index_data.state + 1;
		END_IF
	3:
		index_data.slot_index := index_data.slot_index_nearest;
		index_data.is_home_ing := TRUE;
		index_data.state := 101;
	//index
	101:
		IF AZ_power.Status THEN
			index_data.real_position := index_data.ecd_sing / index_data.ecd_reso;
			index_data.soft_position := AZ.fActPosition / index_data.ecd_reso;
			index_data.offset := index_data.real_position - index_data.soft_position;
			index_data.target_position := INT_TO_LREAL(index_data.slot_index) / INT_TO_LREAL(index_data.slot_count) - index_data.offset; 
			AZ_mabs.Velocity := index_data.ecd_reso * (index_data.feed_rpm / 60.0);
			AZ_mabs.Acceleration := AZ_mabs.Velocity / 0.05;
			AZ_mabs.Deceleration := AZ_mabs.Velocity / 0.05;
			IF index_data.is_home_ing OR index_data.vibrate_distance <= 0.0 THEN
				AZ_mabs.Position := index_data.target_position * index_data.ecd_reso;
				index_data.is_home_ing := FALSE;
				index_data.state := 102;
			ELSE
				AZ_mabs.Position := WRAP(value:= index_data.soft_position - index_data.vibrate_distance, v_min:= 0.0, v_max:= 1.0) * index_data.ecd_reso;
				index_data.state := 151;
			END_IF
			AZ_mabs.Execute := TRUE;
		END_IF
	102:
		IF AZ_mabs.Done THEN
			AZ_mabs.Execute := FALSE;
			index_data.state := 154;
		END_IF
	//back
	151:
		IF AZ_mabs.Done THEN
			AZ_mabs.Execute := FALSE;
			index_data.state := index_data.state + 1;
		END_IF
	152:
		IF AZ_power.Status THEN 
			AZ_mabs.Position := index_data.target_position * index_data.ecd_reso;
			AZ_mabs.Execute := TRUE;
			index_data.state := index_data.state + 1;
		END_IF
	153:
		IF AZ_mabs.Done THEN
			AZ_mabs.Execute := FALSE;
			index_data.state := index_data.state + 1;
		END_IF
	154:
		index_data.end_timer(IN:= , PT:= , Q=> , ET=> );
		IF NOT index_data.end_timer.IN THEN
			index_data.end_timer.IN := TRUE;
			index_data.end_timer.PT := INT_TO_TIME(index_data.end_delay);
		END_IF
		IF index_data.end_timer.Q THEN
			index_data.slot_index := (index_data.slot_index + 1) MOD index_data.slot_count;
			index_data.state := 100;
			index_data.end_timer.IN := FALSE;
		END_IF
END_CASE
END_ACTION

ACTION work:
CASE work_data.state OF
	1:
		work_data.end_timer.IN := FALSE;
		work_data.state := work_data.state + 1;
	2:
		tap_data.state := 0;
		work_data.state := work_data.state + 1;
	3:
		gear_data.state := 1;
		work_data.state := work_data.state + 1;
	4:
		IF gear_data.state = 0 THEN
			gear_data.state := 101;
			work_data.state := work_data.state + 1;
		END_IF
	5:
		IF gear_data.state = 200 THEN
			index_data.state := 0;
			AZ_power.bRegulatorOn := FALSE;
			work_data.state := work_data.state + 1;
		END_IF
	6:
		work_data.state := 0;
	//home
	101:
		IF tap_data.state = 0 THEN
			tap_data.state := 1;
			work_data.state := work_data.state + 1;
		END_IF
	102:
		IF tap_data.state = 100 THEN
			work_data.state := work_data.state + 1;
		END_IF
	103:
		IF index_data.state = 0 THEN
			index_data.state := 1;
			work_data.state := work_data.state + 1;
		END_IF
	104:
		IF index_data.state = 100 THEN
			work_data.state := 200;
		END_IF
	//1 cycle	
	201:
		IF index_data.state = 100 THEN
			tap_data.state := 101;
			work_data.state := work_data.state + 1;
		END_IF
	202:
		IF tap_data.state = 100 THEN
			index_data.state := 101;
			work_data.state := work_data.state + 1;
		END_IF
	203:
		IF index_data.state = 100 THEN
			work_data.state := work_data.state + 1;
		END_IF
	204:
		work_data.end_timer(IN:= , PT:= , Q=> , ET=> );
		IF NOT work_data.end_timer.IN THEN
			work_data.end_timer.IN := TRUE;
			work_data.end_timer.PT := INT_TO_TIME(work_data.end_delay);
		END_IF
		IF work_data.end_timer.Q THEN
			work_data.state := 200;
			work_data.end_timer.IN := FALSE;
		END_IF
END_CASE
END_ACTION

METHOD WRAP : LREAL
VAR_INPUT
	value: LREAL;
	v_min: LREAL;
	v_max: LREAL;
END_VAR
VAR
	range: LREAL;
END_VAR
range := v_max - v_min;
IF ABS(range) < 1E-8 THEN
	WRAP := v_min;
ELSE
	WRAP := value - (range * TRUNC((value - v_min) / range));
	IF ABS(WRAP - v_max) < 1e-8 THEN
		WRAP := v_min;
	END_IF
END_IF
END_METHOD

END_PROGRAM

// Device/Application/Visualization
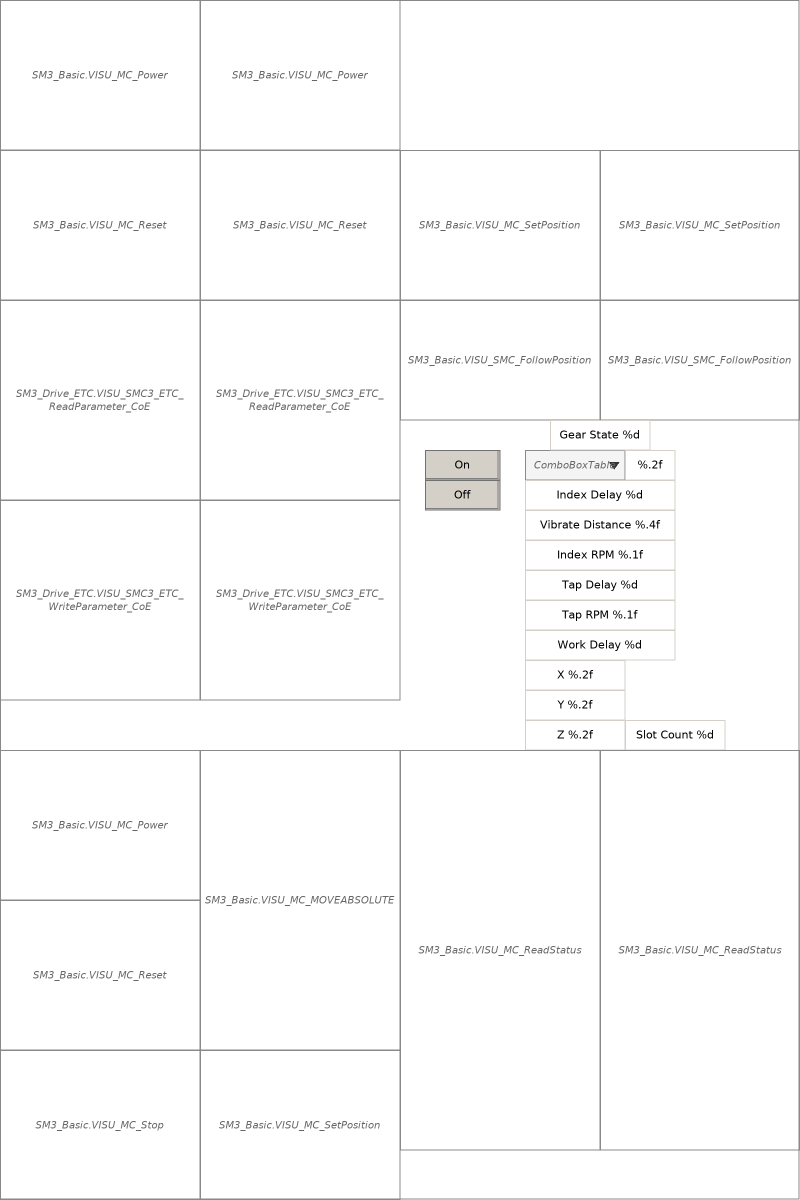
VISUALIZATION Visualization  // 800x1200
    Frame (0,0 200x150)
        shows SM3_Basic.VISU_MC_Power(m_Input_FB := main.AX_power)
    Frame (200,0 200x150)
        shows SM3_Basic.VISU_MC_Power(m_Input_FB := main.AY_power)
    Frame (0,150 200x150)
        shows SM3_Basic.VISU_MC_Reset(m_Input_FB := main.AX_reset)
    Frame (200,150 200x150)
        shows SM3_Basic.VISU_MC_Reset(m_Input_FB := main.AY_reset)
    Frame (0,300 200x200)
        shows SM3_Drive_ETC.VISU_SMC3_ETC_ReadParameter_CoE(m_Input_FB := main.AX_read)
    Frame (0,500 200x200)
        shows SM3_Drive_ETC.VISU_SMC3_ETC_WriteParameter_CoE(m_Input_FB := main.AX_write)
    Frame (200,300 200x200)
        shows SM3_Drive_ETC.VISU_SMC3_ETC_ReadParameter_CoE(m_Input_FB := main.AY_read)
    Frame (200,500 200x200)
        shows SM3_Drive_ETC.VISU_SMC3_ETC_WriteParameter_CoE(m_Input_FB := main.AY_write)
    Frame (400,150 200x150)
        shows SM3_Basic.VISU_MC_SetPosition(m_Input_FB := main.AX_set_position)
    Frame (600,150 200x150)
        shows SM3_Basic.VISU_MC_SetPosition(m_Input_FB := main.AY_set_position)
    Frame (400,300 200x120)
        shows SM3_Basic.VISU_SMC_FollowPosition(m_Input_FB := main.AX_follow)
    Textfield (525,660 100x30), "X %.2f", text variable: AX.fActPosition
    Textfield (525,690 100x30), "Y %.2f", text variable: AY.fActPosition
    ComboBoxTable (525,450 100x30), variable: main.gear_data.ratio_array_index, data array: main.gear_data.ratio_array
        p1014161805: 14 - 0 + 1
        p3854506369: main.gear_data.ratio_array[INDEX]
    Textfield (625,450 50x30), "%.2f", text variable: main.gear_data.ratio_target
    Frame (0,750 200x150)
        shows SM3_Basic.VISU_MC_Power(m_Input_FB := main.AZ_power)
    Frame (0,900 200x150)
        shows SM3_Basic.VISU_MC_Reset(m_Input_FB := main.AZ_reset)
    Frame (0,1050 200x150)
        shows SM3_Basic.VISU_MC_Stop(m_Input_FB := main.AZ_stop)
    Frame (200,750 200x300)
        shows SM3_Basic.VISU_MC_MOVEABSOLUTE(m_Input_FB := main.AZ_mabs)
    Frame (200,1050 200x150)
        shows SM3_Basic.VISU_MC_SetPosition(m_Input_FB := main.AZ_set_position)
    Textfield (525,720 100x30), "Z %.2f", text variable: AZ.fActPosition
    Textfield (525,480 150x30), "Index Delay %d", text variable: main.index_data.end_delay
        OnMouseClick: write the text variable via Default, min 10, max 5000
    Textfield (625,720 100x30), "Slot Count %d", text variable: main.index_data.slot_count
        OnMouseClick: write the text variable via Default, min 3, max 16
    Textfield (525,570 150x30), "Tap Delay %d", text variable: main.tap_data.end_delay
        OnMouseClick: write the text variable via Default, min 10, max 5000
    Textfield (525,630 150x30), "Work Delay %d", text variable: main.work_data.end_delay
        OnMouseClick: write the text variable via Default, min 10, max 5000
    Textfield (525,600 150x30), "Tap RPM %.1f", text variable: main.tap_data.feed_rpm
        OnMouseClick: write the text variable via Default, min 300, max 3000
    Textfield (525,510 150x30), "Vibrate Distance %.4f", text variable: main.index_data.vibrate_distance
        OnMouseClick: write the text variable via Default, min 0, max 0.05
    Textfield (525,540 150x30), "Index RPM %.1f", text variable: main.index_data.feed_rpm
        OnMouseClick: write the text variable via Default, min 1, max 180
    Frame (600,300 200x120)
        shows SM3_Basic.VISU_SMC_FollowPosition(m_Input_FB := main.AY_follow)
    Textfield (550,420 100x30), "Gear State %d", text variable: main.gear_data.state
        OnMouseClick: write the text variable via Default, min 0, max 1000
    Button (425,450 75x30), "On", pressed state: main.button_data.on
        toggle main.button_data.on
    Button (425,480 75x30), "Off", pressed state: main.button_data.off
        toggle main.button_data.off
    Frame (400,750 200x400)
        shows SM3_Basic.VISU_MC_ReadStatus(m_Input_FB := main.AX_status)
    Frame (600,750 200x400)
        shows SM3_Basic.VISU_MC_ReadStatus(m_Input_FB := main.AY_status)
END_VISUALIZATION
